Staubli VAL3: StaubliCalTool7.pjx

--- StaubliCalTool7.pjx ---
Parameters version=s7.6.4 stackSize=5000 millimeterUnit=true
Program file=AdjustOffset.pgx
Program file=calSphereCenter.pgx
Program file=calTool.pgx
Program file=CheckPosEqual.pgx
Program file=CheckTraj.pgx
Program file=ClsPage.pgx
Program file=Control_YesNo.pgx
Program file=InitData.pgx
Program file=interpolatePos.pgx
Program file=Language.pgx
Program file=ListMove.pgx
Program file=ListMsg.pgx
Program file=ListMsgC.pgx
Program file=ListMsgE.pgx
Program file=ListPop.pgx
Program file=ListPopC.pgx
Program file=ListPopE.pgx
Program file=Main.pgx
Program file=ReadMe.pgx
Program file=setTool.pgx
Program file=splitUp.pgx
Program file=start.pgx
Program file=Step1_Mount.pgx
Program file=Step2_Teach.pgx
Program file=Step3_AdjustXY.pgx
Program file=Step4_AdjustZ.pgx
Program file=Step5_Test.pgx
Program file=stop.pgx
Program file=Version20141125.pgx
Program file=xyPut.pgx
Data file=StaubliCalTool7.dtx

--- calTool.pgx ---
program CalTool(string x_sCalTool (dimensions=1))
  local num l_nDistance
  local trsf l_trFlange
  local trsf l_trTCP
  local trsf l_trZ
begin
  switch x_sCalTool
    case "CalTool1"
      call SplitUp()
      call CalSphereCenter(nS1[1],nS2[1],nS3[1],nS4[1],nS1[2],nS2[2],nS3[2],nS4[2],nS1[3],nS2[3],nS3[3],nS4[3])
      if ((nScX==9999.9999) or (nScY==9999.9999) or (nScZ==9999.9999))
        call InitData()
        call ListPop("DeviationIsTooLarge")
      else
        l_trFlange={0,0,0,0,0,0}
        l_trTCP={0,0,0,0,0,0}
        l_trFlange=p1_1.trsf
        if sMount=="floor"
          l_trTCP={nScX,nScY,nScZ,0,180,0}
        elseIf sMount=="ceiling"
          l_trTCP={nScX,nScY,nScZ,0,0,0}
        endIf
        tTool1.trsf=!l_trFlange*l_trTCP
      endIf
      call ListPop("SaveInTool1")
    break

    case "CalTool2_2"
      l_trFlange={0,0,0,0,0,0}
      l_trTCP={0,0,0,0,0,0}
      nScX=(p2_2_1.trsf.x+p2_2_2.trsf.x)/2
      nScY=(p2_2_1.trsf.y+p2_2_2.trsf.y)/2
      nScZ=(p2_2_1.trsf.z+p2_2_2.trsf.z)/2
      //
      l_trFlange=p2_2_1.trsf*!tTool.trsf
      if sMount=="floor"
        l_trTCP={nScX,nScY,nScZ,0,180,0}
      elseIf sMount=="ceiling"
        l_trTCP={nScX,nScY,nScZ,0,0,0}
      endIf
      tTool2.trsf=!l_trFlange*l_trTCP
      //
      tTool2.trsf.rx=tTool1.trsf.rx
      tTool2.trsf.ry=tTool1.trsf.ry
      tTool2.trsf.rz=tTool1.trsf.rz
      call ListPop("SaveInTool2")
    break
    case "CalTool2_3"
      l_trFlange={0,0,0,0,0,0}
      l_trTCP={0,0,0,0,0,0}
      nScX=p2_3_2.trsf.x+p2_3_3.trsf.x-p2_3_1.trsf.x
      nScY=p2_3_2.trsf.y+p2_3_3.trsf.y-p2_3_1.trsf.y
      nScZ=p2_3_2.trsf.z+p2_3_3.trsf.z-p2_3_1.trsf.z
      //
      l_trFlange=p2_3_1.trsf*!tTool.trsf
      if sMount=="floor"
        l_trTCP={nScX,nScY,nScZ,0,180,0}
      elseIf sMount=="ceiling"
        l_trTCP={nScX,nScY,nScZ,0,0,0}
      endIf
      tTool2.trsf=!l_trFlange*l_trTCP
      //
      tTool2.trsf.rx=tTool1.trsf.rx
      tTool2.trsf.ry=tTool1.trsf.ry
      tTool2.trsf.rz=tTool1.trsf.rz
      call ListPop("SaveInTool2")
    break
    case "CalTool3"
      l_nDistance=distance(p3_1,p3_2)
      if nMount==1 or nMount==-1
        if p3_1.trsf.z<p3_2.trsf.z
          l_trZ={0,0,-l_nDistance*nMount,0,0,0}
        else
          l_trZ={0,0,l_nDistance*nMount,0,0,0}
        endIf
        tTool3.trsf=tTool.trsf*l_trZ
        tTool3.trsf.rx=tTool1.trsf.rx
        tTool3.trsf.ry=tTool1.trsf.ry
        tTool3.trsf.rz=tTool1.trsf.rz
        call ListPop("SaveInTool3")
      else
        call ListPop("SetMounting")
      endIf
    break
  endSwitch
end

--- InitData.pgx ---
program InitData()
  local num l_nI
begin
  setTextMode(0)
  $jogPage(false)
  $jogContext(flange,world,0)
  sLanguge="Chinese"
  bFinish=false
  bUpLoad=false
  sTool="flange"
  sMount="floor"
  nMount=1
  //
  nOffsetX=0
  nOffsetY=0
  nOffsetZ=0
  nOffsetRx=0
  nOffsetRy=0
  nOffsetRz=0
  //
  mNomSpeed.blend=Cartesian
  mNomSpeed.leave=mNomSpeed.reach=50
  mSpeed.blend=Cartesian
  mSpeed.leave=mSpeed.reach=0
  mSlow.blend=Cartesian
  mSlow.leave=mSlow.reach=0
  mSlow.vel=2
  //
  cConfigSame={ssame,esame,wsame}
  //
  //  tTool.trsf={0,0,0,0,0,0}
  //  tTool1.trsf={0,0,0,0,0,0}
  //  tTool2.trsf={0,0,0,0,0,0}
  //  tTool3.trsf={0,0,0,0,0,0}
  //
  p1_1.trsf={0,0,0,0,0,0}
  p1_1.config={ssame,esame,wsame}
  p1_2.trsf={0,0,0,0,0,0}
  p1_2.config={ssame,esame,wsame}
  p1_3.trsf={0,0,0,0,0,0}
  p1_3.config={ssame,esame,wsame}
  p1_4.trsf={0,0,0,0,0,0}
  p1_4.config={ssame,esame,wsame}
  p2_2_1.trsf={0,0,0,0,0,0}
  p2_2_1.config={ssame,esame,wsame}
  p2_2_2.trsf={0,0,0,0,0,0}
  p2_2_2.config={ssame,esame,wsame}
  p2_3_1.trsf={0,0,0,0,0,0}
  p2_3_1.config={ssame,esame,wsame}
  p2_3_2.trsf={0,0,0,0,0,0}
  p2_3_2.config={ssame,esame,wsame}
  p2_3_3.trsf={0,0,0,0,0,0}
  p2_3_3.config={ssame,esame,wsame}
  p3_1.trsf={0,0,0,0,0,0}
  p3_1.config={ssame,esame,wsame}
  p3_2.trsf={0,0,0,0,0,0}
  p3_2.config={ssame,esame,wsame}
  //
  bTeach1_1=false
  bTeach1_2=false
  bTeach1_3=false
  bTeach1_4=false
  bTeach2_2_1=false
  bTeach2_2_2=false
  bTeach2_3_1=false
  bTeach2_3_2=false
  bTeach2_3_3=false
  bTeach3_1=false
  bTeach3_2=false
  //
  nScX=nScY=nScZ=0
  for l_nI=0 to 3
    nS1[l_nI]=nS2[l_nI]=nS3[l_nI]=nS4[l_nI]=0
  endFor
end

--- ListMove.pgx ---
program ListMove(string x_sM (dimensions=1))
  local bool l_bA
  local bool l_bB
  local bool l_bEqual
  local frame l_fFrame
  local joint l_jJoint
  local trsf l_trR
begin
  switch x_sM
    case "align"
      resetMotion()
      call ListPop("PressMoveHoldToAlign")
      pA.trsf={0,0,0,0,0,0}
      pA=here(tTool,world)
      pA.trsf=align(pA.trsf,world.trsf)
      movel(pA,tTool,mSpeed)
      waitEndMove()
      resetMotion()
      call ListPop("CompletedAlign")
    break
    case "GoBackP2_2_1"
      if p2_2_1.trsf!={0,0,0,0,0,0}
        resetMotion()
        call CheckPosEqual(p2_2_1,l_bEqual)
        if l_bEqual==false
          call ListPop("PressMoveHoldToGoBack")
          call interpolatePos(here(tTool,world),p2_2_1)
          call ListPop("CompletedGoBack")
        endIf
      else
        call ListPop("CantGoBack")
      endIf
    break
    case "Rz+180P2_2_1"
      resetMotion()
      pA.trsf={0,0,0,0,0,0}
      pB.trsf={0,0,0,0,0,0}
      l_trR={0,0,0,0,0,90}
      pA.trsf=p2_2_1.trsf*l_trR
      pA.config=cConfigSame
      pB.trsf=pA.trsf*l_trR
      pB.config=cConfigSame
      call CheckTraj(p2_2_1,pA,l_bA)
      call CheckTraj(pA,pB,l_bB)
      if l_bA==true and l_bB==true
        movel(pA,tTool,mSpeed)
        movel(pB,tTool,mSpeed)


        waitEndMove()
        call ListPop("CompletedMove")
      endIf
    break
    case "Rz-180P2_2_1"
      resetMotion()
      pA.trsf={0,0,0,0,0,0}
      pB.trsf={0,0,0,0,0,0}
      l_trR={0,0,0,0,0,-90}
      pA.trsf=p2_2_1.trsf*l_trR
      pA.config=cConfigSame
      pB.trsf=pA.trsf*l_trR
      pB.config=cConfigSame
      call CheckTraj(p2_2_1,pA,l_bA)
      call CheckTraj(pA,pB,l_bB)
      if l_bA==true and l_bB==true
        movel(pA,tTool,mSpeed)
        movel(pB,tTool,mSpeed)
        waitEndMove()
        call ListPop("CompletedMove")
      endIf
    break
    case "GoBackP2_3_1"
      if p2_3_1.trsf!={0,0,0,0,0,0}
        resetMotion()
        call CheckPosEqual(p2_2_1,l_bEqual)
        if l_bEqual==false
          call ListPop("PressMoveHoldToGoBack")
          call interpolatePos(here(tTool,world),p2_3_1)
          call ListPop("CompletedGoBack")
        endIf
      else
        call ListPop("CantGoBack")
      endIf
    break
    case "Rz+60P2_3_1"
      resetMotion()
      call ListPop("PressMoveHoldToMove")
      pA.trsf={0,0,0,0,0,0}
      l_trR={0,0,0,0,0,60}
      pA.trsf=p2_3_1.trsf*l_trR
      pA.config=cConfigSame
      call CheckTraj(p2_3_1,pA,l_bA)
      if l_bA==true
        movel(pA,tTool,mSpeed)
        waitEndMove()
        call ListPop("CompletedMove")
      endIf
    break
    case "Rz-60P2_3_1"
      resetMotion()
      call ListPop("PressMoveHoldToMove")
      pA.trsf={0,0,0,0,0,0}
      l_trR={0,0,0,0,0,-60}
      pA.trsf=p2_3_1.trsf*l_trR
      pA.config=cConfigSame
      call CheckTraj(p2_3_1,pA,l_bA)
      if l_bA==true
        movel(pA,tTool,mSpeed)
        waitEndMove()
        call ListPop("CompletedMove")
      endIf
    break
    case "GoBackP3_1"
      if p3_1.trsf!={0,0,0,0,0,0}
        resetMotion()
        call CheckPosEqual(p3_1,l_bEqual)
        if l_bEqual==false
          call ListPop("PressMoveHoldToGoBack")
          pB=appro(p3_1,{0,0,-10,0,0,0})
          movel(pB,tTool,mSpeed)
          movel(p3_1,tTool,mSlow)
          call ListPop("CompletedGoBack")
        endIf
      else
        call ListPop("CantGoBack")
      endIf
    break

    case "Rx+60P3_1"
      resetMotion()
      call ListPop("PressMoveHoldToMove")
      pA.trsf={0,0,0,0,0,0}
      l_fFrame.trsf={p3_1.trsf.x,p3_1.trsf.y,p3_1.trsf.z,0,0,0}
      l_trR={0,0,0,60,0,0}
      pA.trsf=l_fFrame.trsf*l_trR*!l_fFrame.trsf*p3_1.trsf
      pB=appro(p3_1,{0,0,-10,0,0,0})
      pA.config=cConfigSame
      pB.config=cConfigSame
      call CheckTraj(p3_1,pB,l_bA)
      call CheckTraj(pB,pA,l_bB)
      if l_bA==true and l_bB==true
        movel(pB,tTool,mSpeed)
        movel(pA,tTool,mSpeed)
        waitEndMove()
        call ListPop("CompletedMove")
      endIf
    break
    case "Ry+60P3_1"
      resetMotion()
      call ListPop("PressMoveHoldToMove")
      pA.trsf={0,0,0,0,0,0}
      l_fFrame.trsf={p3_1.trsf.x,p3_1.trsf.y,p3_1.trsf.z,0,0,0}
      l_trR={0,0,0,0,60,0}
      pA.trsf=l_fFrame.trsf*l_trR*!l_fFrame.trsf*p3_1.trsf
      pB=appro(p3_1,{0,0,-10,0,0,0})
      pA.config=cConfigSame
      pB.config=cConfigSame
      call CheckTraj(p3_1,pB,l_bA)
      call CheckTraj(pB,pA,l_bB)
      if l_bA==true and l_bB==true
        movel(pB,tTool,mSpeed)
        movel(pA,tTool,mSpeed)
        waitEndMove()
        call ListPop("CompletedMove")
      endIf
    break
  endSwitch
end

--- ListMsg.pgx ---
program ListMsg(bool x_bRefresh (dimensions=1), string x_sS (dimensions=1))
begin
  switch sLanguge
    case "English"
      call ListMsgE(x_bRefresh,x_sS)
    break
    case "Chinese"
      call ListMsgC(x_bRefresh,x_sS)
    break
  endSwitch
end

--- ListPopC.pgx ---
program ListPopC(string x_sS (dimensions=1))
begin
  switch x_sS
    case "OffsetDone"
      popUpMsg("偏差设置完成")
    break
    case "Offset"
      popUpMsg("填入偏差后请按回车确认")
    break
    case "Floor"
      popUpMsg("当前安装方式已设置成floor")
    break
    case "Ceiling"
      popUpMsg("当前安装方式已设置成ceiling")
    break
    case "First"
      popUpMsg("第1点记录完成")
    break
    case "Second"
      popUpMsg("第2点记录完成")
    break
    case "Third"
      popUpMsg("第3点记录完成")
    break
    case "Fourth"
      popUpMsg("第4点记录完成")
    break
    case "FRP"
      popUpMsg("请先记录点")
    break
    case "CantSwitchTool2"
      popUpMsg("不能切换tTool2!请先标定tTool1!")
    break
    case "CantSwitchTool3"
      popUpMsg("不能切换tTool3!请先标定tTool2!")
    break
    case "DeviationIsTooLarge"
      popUpMsg("偏差过大!请重新记录4点!")
    break
    case "SaveInTool1"
      popUpMsg("工具参数保存在tTool1")
    break
    case "SaveInTool2"
      popUpMsg("工具参数保存在tTool2")
    break
    case "SaveInTool3"
      popUpMsg("工具参数保存在tTool3")
    break
    case "SetMounting"
      popUpMsg("请先设置机器人安装方式")
    break
    case "PressMoveHoldToAlign"
      popUpMsg("请按Move/Hold键对齐")
    break
    case "PressMoveHoldToGoBack"
      popUpMsg("请按Move/Hold键重置")
    break
    case "PressMoveHoldToMove"
      popUpMsg("请按Move/Hold键移动")
    break
    case "CompletedAlign"
      popUpMsg("对齐完成")
    break
    case "CompletedGoBack"
      popUpMsg("重置完成")
    break
    case "CompletedMove"
      popUpMsg("移动完成")
    break
    case "CantMove"
      popUpMsg("不可到达！请重新记录第1点")
    break
    case "CantGoBack"
      popUpMsg("不可重置！请首先记录第1点")
    break
    case "CompletedUpLoad"
      popUpMsg("工具上传完成")
    break
    case "EndOfProgram"
      popUpMsg("欢迎使用史陶比尔软件")
    break
  endSwitch
end

--- ReadMe.pgx ---
program ReadMe()
begin
  //-----------------------------------------------------------------------
  //                    史陶比尔工具标定程序
  //
  //主要功能：不拆激光头实现工具位置与姿态的标定和修正
  //          标定精度可以达到已有的拆工具方法的标定精度
  //          工具标定误差小于1mm
  //工具数据：tTool1初次标定后的工具值，此时工具中心点与激光头存在一定距离误差
  //          tTool2修正xy后的工具值，此时工具中心点与激光头基本在同一轴线
  //          tTool3修正z后的工具值，此时工具中心点与激光头基本重合
  //功能介绍:
  //     安装方式：置顶或者置地
  //
  //     标定工具：flange记录4点计算得到工具tTool1
  //
  //     修正工具XY：tTool1记录2或3点修正得到工具tTool2
  //         两点法180°修正工具XY(优先选择此方法，比较准确)
  //         三点法±60°修正工具XY(如果toolRz不能旋转180°选择此方法)
  //
  //     修正工具Z：tTool2记录2点修正得到工具tTool3
  //
  //     测试工具：可以切换、对齐、修改当前工具
  //
  //
  //补充说明：这里的修正指的是对工具TCP位置的修正，而不是工具姿态的修正
  //          一个TCP值可以用一个4x4矩阵来表达，如果用X-Y-Z欧拉角的方式提取6个参数{x、y、z、rx、ry、rz}
  //          x、y、z是唯一解，rx、ry、rz存在两组解，其中rz可以是任意值
  //
  //
  //                                                      2012.8.16   张华君
  //
  // 修改:可以使用已标定的工具继续标定自身                2012.9.3    张华君
  //
  // 修改:重写HMI                                         2012.11.21   张华君
  //
  // 修改:1.修正工具再标定的Bug
  //      2.重新程序框架，增加英文界面                    2013.3.21    张华君
  //
  // 修改:增加计算点是否可达的判断                        2013.4.25    张华君
  //
  // 修改:1.增加手动微调工具值的功能                      2013.5.13    张华君
  //      2.title显示当前操作步骤
  //      3.标定结果合并到测试工具页面当中
  //
  // 修改：2点法180°修正XY时，修正目标点不能预判是否能到达       2014.06.13 张华君
  //
  // 修改: AdjustXY调节推出的页面报错问题                         2014.11.25 张华君
  //--------------------------------------------------------------------
end

--- Step1_Mount.pgx ---
program Step1_Mount()
  local bool l_bOut
  local num l_nKey
begin
  call ListMsg(true,"HMImount")
  l_bOut=false
  while !l_bOut
    do
      l_nKey=get()-270
    until l_nKey==1 or l_nKey==2 or l_nKey==7 or l_nKey==-15
    switch l_nKey
      case 1
        nMount=1
        sMount="floor"
        call ListMsg(true,"HMImount")
        call ListPop("Floor")
      break
      case 2
        nMount=-1
        sMount="ceiling"
        call ListMsg(true,"HMImount")
        call ListPop("Ceiling")
      break
      case 7,-15
        wait(getKey()==-1)
        call ListMsg(true,"HMImain")
        l_bOut=true
      break
    endSwitch
  endWhile
end
